// Mitsubishi GX Works2 project: example_q   PLC: Q00J

PROGRAM MAIN
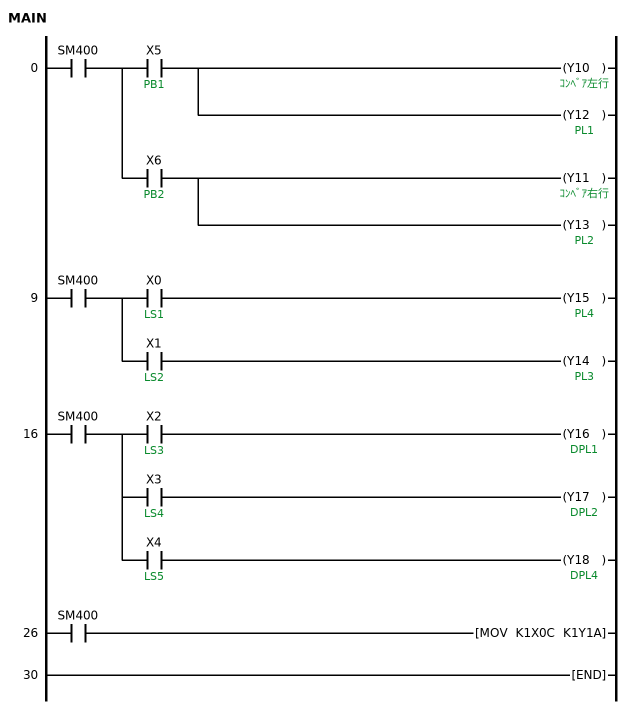
0     LD      SM400
      MPS
      AND     X5  ; PB1
      OUT     Y10  ; ｺﾝﾍﾞｱ左行
      OUT     Y12  ; PL1
      MPP
      AND     X6  ; PB2
      OUT     Y11  ; ｺﾝﾍﾞｱ右行
      OUT     Y13  ; PL2
9     LD      SM400
      MPS
      AND     X0  ; LS1
      OUT     Y15  ; PL4
      MPP
      AND     X1  ; LS2
      OUT     Y14  ; PL3
16    LD      SM400
      MPS
      AND     X2  ; LS3
      OUT     Y16  ; DPL1
      MRD
      AND     X3  ; LS4
      OUT     Y17  ; DPL2
      MPP
      AND     X4  ; LS5
      OUT     Y18  ; DPL4
26    LD      SM400
      MOV     K1X0C K1Y1A  ; DSW1 / DPL10
30    END
END_PROGRAM
